PROGRAM MAIN
VAR
	fbMessanger 			: FB_Messenger;
	arstHTTP_Messages_In 	: ARRAY[0..2] OF ST_HTTP_MESSAGE;
	arstHTTP_Messages_Out 	: ARRAY[0..2] OF ST_HTTP_MESSAGE;
	arstStruct 				: ARRAY [0..999] OF ST_STRUCT;
	arstCat 				: ARRAY [0..99] OF ST_CAT;
END_VAR
VAR CONSTANT
	arstRequest_Line : ARRAY[0..2] OF ST_REQUEST_LINE :=
									[ 
										( eMethod := E_METHOD.GET, sURI := '/brands/toyota.html', sProtocol := 'HTTP/1.1'),
										( eMethod := E_METHOD.GET, sURI := '/brands/suzuki.html', sProtocol := 'HTTP/1.1'),
										( eMethod := E_METHOD.GET, sURI := '/_/mss/boq-one-google/_/js', sProtocol := 'HTTP/1.1')
									];
	arstHeader_Fields : ARRAY[0..2] OF ST_HEADER_FIELDS := 
									[
										(sHost := 'www.cars.com', sAccept := 'text/html text/plain image/gif image/jpeg', sAccept_Language := 'en-GB', sAccept_Encoding := 'gzip, deflate', sUser_Agent := 'Safari/537.36'),
										(sHost := 'www.cars.com', sAccept := 'text/html text/plain image/gif image/jpeg', sAccept_Language := 'en-US,en;q=0.9', sAccept_Encoding := 'gzip, deflate', sUser_Agent := 'Chrome/102.0.5005.124'),
										(sHost := 'www.gstatic.com', sAccept := '*/*', sAccept_Language := 'en-US,en;q=0.9', sAccept_Encoding := 'gzip, deflate, br', sUser_Agent := 'Mozilla/5.0')
									];
END_VAR

arstHTTP_Messages_Out[0].stRequest_Line := arstRequest_Line[0];
arstHTTP_Messages_Out[0].stHeader_Fields := arstHeader_Fields[0];

arstHTTP_Messages_Out[1].stRequest_Line := arstRequest_Line[1];
arstHTTP_Messages_Out[1].stHeader_Fields := arstHeader_Fields[1];

arstHTTP_Messages_Out[2].stRequest_Line := arstRequest_Line[2];
arstHTTP_Messages_Out[2].stHeader_Fields := arstHeader_Fields[2];

END_PROGRAM

(* stored: Version 1.1.0.1, ProductVersion 3.1.4024.4
   POU MAIN: Id {ef0ca126-29ac-4ca2-946e-77fc5278adf9}, SpecialFunc None *)
